// TIA Portal V20 export
VAR_GLOBAL   // PLC tag table "Constantes del Nucleo 2021"
END_VAR
VAR_GLOBAL CONSTANT   // user constants
   CTE_MaxArrayConversion : UInt := 500;
END_VAR
